FUNCTION_BLOCK PUBLIC FB_Device EXTENDS FB_ComponentBase
VAR_INPUT
	// IO reference
	stIn		: ST_DeviceIn;
	//stIO : REFERENCE TO ST_DeviceIO;
END_VAR
VAR_OUTPUT
	bOut		: BOOL;
	fValue		: LREAL;
	stOut		: ST_DeviceOut;
END_VAR
VAR
	// private var's
	bEnable : BOOL;
END_VAR

bOut := stOut.bRun;
fValue := stout.fValue;

PROPERTY PUBLIC Enable : BOOL
GET
Enable := bEnable;
END_GET
SET
bEnable := Enable;
END_SET
END_PROPERTY

METHOD PUBLIC M_Off : BOOL;
VAR_INPUT
END_VAR
stOut.bRun := FALSE;
M_Off := TRUE;
END_METHOD

METHOD PUBLIC M_On : BOOL;
VAR_INPUT
END_VAR
IF bEnable THEN
	stOut.bRun := TRUE;
	M_On := TRUE;
END_IF
END_METHOD

METHOD M_Reset : BOOL
VAR_INPUT
END_VAR
M_Reset := TRUE;
END_METHOD

{attribute 'monitoring' := 'call'}
PROPERTY PUBLIC Value : LREAL
GET
Value := stOut.fValue;
END_GET
SET
stOut.fValue := Value;
END_SET
END_PROPERTY

END_FUNCTION_BLOCK

(* stored: Version 1.1.0.1, ProductVersion 3.1.4024.12
   POU FB_Device: Id {7f23a655-b176-447d-80d0-4d1a4ddd490b}, SpecialFunc None
   Property Enable: Id {e4721e20-53b4-4670-87fa-30bbcc95656d}
   Get Get: Id {9727f9ac-59df-43d2-bb46-57830436bd38}
   Set Set: Id {77c89f51-8570-4e1b-a012-6e54f8f56d9c}
   Method M_Off: Id {a13597b7-8b8a-4945-8888-edf7b53cfaa2}
   Method M_On: Id {f17dde1d-ffa4-4d42-bf9e-d7ad881568ae}
   Method M_Reset: Id {57fa2749-3f58-4840-a0b8-f25232cbf356}
   Property Value: Id {0585073b-32fd-44b5-8171-bd856093f69b}
   Get Get: Id {cacae9ac-2971-420a-a48b-8fd2f86e8955}
   Set Set: Id {a9351200-a99a-4427-b7f4-b8a36d069494} *)
